GLOBALCONSTANTS myPorts_espnow (* Global constants *)
  (* Standard: 61499-1 *)
  (* Version 1.0, 2023-10-22, franz *)
  VAR_GLOBAL CONSTANT
    PORT_0_espnow : WSTRING := "fbdk[].espnow[239.0.0.1:61000]";
    PORT_1_espnow : WSTRING := "fbdk[].espnow[239.0.0.1:61001]";
    PORT_2_espnow : WSTRING := "fbdk[].espnow[239.0.0.1:61002]";
    PORT_3_espnow : WSTRING := "fbdk[].espnow[239.0.0.1:61003]";
  END_VAR
END_GLOBALCONSTANTS
